(* Logix 5000 project; controller IPG_2332_07A 1769-L16ER-BB1B rev 34.12; software revision 34.01; part 3 of 4 *)
(* tags used below, declared in another part *)
   Axis_Controller : udt_Zaber_Axis;
   Flash_320mS : BOOL;
   Flash_640mS : BOOL;
   p_Alarmed_Time : String_15;
   p_All_Axis_Home : DINT;
   p_AOI_Cycle_Times : AOI_Cycle_Times;
   p_ASCII_RXID : DINT;
   p_ASCII_TXID : COUNTER;
   p_Axis_ONS : DINT;
   p_Barcode_results_Count_prev : DINT;
   p_BarcodeDone : BOOL;
   p_Cassette_Data : DINT;
   p_Cassette_Data_String : STRING;
   p_CassetteGripper_OUT : BOOL;
   p_CassetteRelease_IN : BOOL;   // Foot Switch
   p_Control : udt_Machine_Control_V2;   // Main Control
   p_Data_Reset : BOOL;
   p_DispenseStart_OUT : BOOL;
   p_DispenseTime : REAL;
   p_Downtime : String_15;
   p_FerruleGripper_OUT : BOOL;
   p_FiberAxis : udt_Zaber_Axis;
   p_FiberAxis_FinalMove_Done : BOOL;
   p_FiberAxis_FinalMoveRel : BOOL;
   p_FiberAxis_FindPos : udt_Station_Sequence;
   p_FiberAxis_InitialMove_Done : BOOL;
   p_FiberAxis_InitialMoveRel : BOOL;
   p_FiberAxis_Move_01_String : STRING;
   p_FiberAxis_Move_02_String : STRING;
   p_FiberGripper_OUT : BOOL;
   p_LED_Ramp : BOOL;
   p_LifeTime_Part_Counter : DINT;
   p_MirrorAxis : udt_Zaber_Axis;
   p_Part_Counter : DINT;
   p_PBLight_Amber_OUT : BOOL;
   p_PBLight_Green_OUT : BOOL;
   p_PBLight_Red_OUT : BOOL;
   p_Sequence : udt_Station_Sequence;
   p_StackLight_Amber_OUT : BOOL;
   p_StackLight_Green_OUT : BOOL;
   p_StackLight_Red_OUT : BOOL;
   p_SyringeAxis : udt_Zaber_Axis;
   p_Uptime : String_15;
   p_Waiting : BOOL;
   p_Waiting_Time : String_15;
   Debug_SDF : DINT;
(* MainProgram_10Ms, continued *)

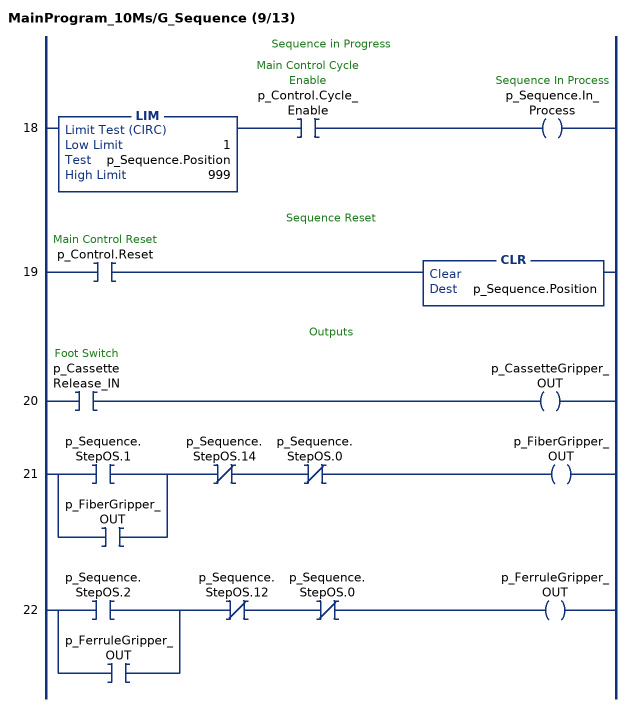
   [picture p43: MainProgram_10Ms/G_Sequence rungs 18-22]
   // Sequence in Progress
   18: LIM(1,p_Sequence.Position,999)XIC(p_Control.Cycle_Enable)OTE(p_Sequence.In_Process);
   // Sequence Reset
   19: XIC(p_Control.Reset)CLR(p_Sequence.Position);
   // Outputs
   20: XIC(p_CassetteRelease_IN)OTE(p_CassetteGripper_OUT);
   21: [XIC(p_Sequence.StepOS.1) ,XIC(p_FiberGripper_OUT) ]XIO(p_Sequence.StepOS.14)XIO(p_Sequence.StepOS.0)OTE(p_FiberGripper_OUT);
   22: [XIC(p_Sequence.StepOS.2) ,XIC(p_FerruleGripper_OUT) ]XIO(p_Sequence.StepOS.12)XIO(p_Sequence.StepOS.0)OTE(p_FerruleGripper_OUT);
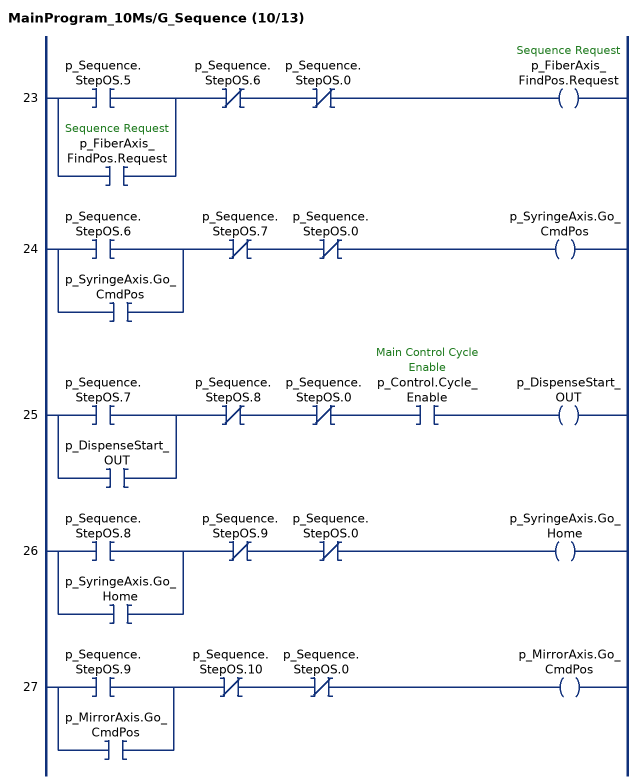
   23: [XIC(p_Sequence.StepOS.5) ,XIC(p_FiberAxis_FindPos.Request) ]XIO(p_Sequence.StepOS.6)XIO(p_Sequence.StepOS.0)OTE(p_FiberAxis_FindPos.Request);
   24: [XIC(p_Sequence.StepOS.6) ,XIC(p_SyringeAxis.Go_CmdPos) ]XIO(p_Sequence.StepOS.7)XIO(p_Sequence.StepOS.0)OTE(p_SyringeAxis.Go_CmdPos);
   25: [XIC(p_Sequence.StepOS.7) ,XIC(p_DispenseStart_OUT) ]XIO(p_Sequence.StepOS.8)XIO(p_Sequence.StepOS.0)XIC(p_Control.Cycle_Enable)OTE(p_DispenseStart_OUT);
   26: [XIC(p_Sequence.StepOS.8) ,XIC(p_SyringeAxis.Go_Home) ]XIO(p_Sequence.StepOS.9)XIO(p_Sequence.StepOS.0)OTE(p_SyringeAxis.Go_Home);
   27: [XIC(p_Sequence.StepOS.9) ,XIC(p_MirrorAxis.Go_CmdPos) ]XIO(p_Sequence.StepOS.10)XIO(p_Sequence.StepOS.0)OTE(p_MirrorAxis.Go_CmdPos);
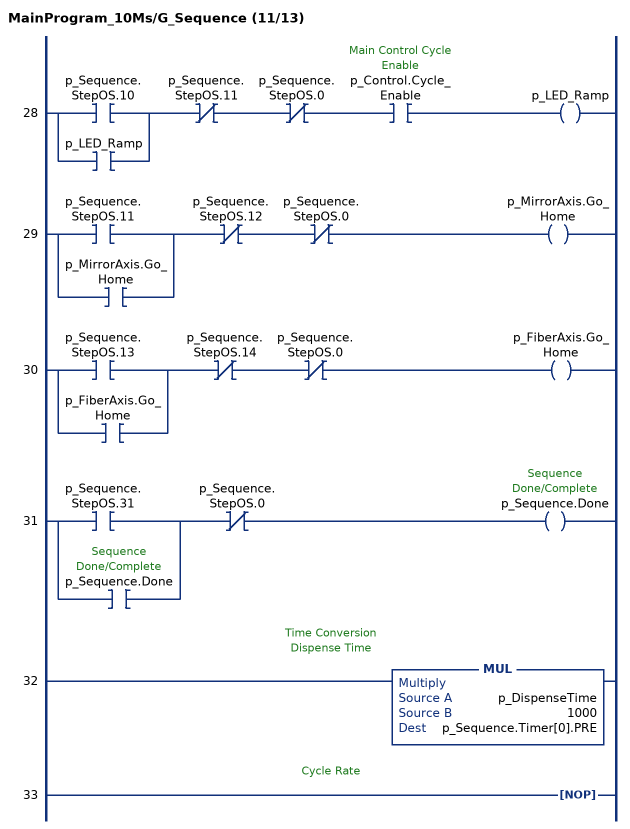
   28: [XIC(p_Sequence.StepOS.10) ,XIC(p_LED_Ramp) ]XIO(p_Sequence.StepOS.11)XIO(p_Sequence.StepOS.0)XIC(p_Control.Cycle_Enable)OTE(p_LED_Ramp);
   29: [XIC(p_Sequence.StepOS.11) ,XIC(p_MirrorAxis.Go_Home) ]XIO(p_Sequence.StepOS.12)XIO(p_Sequence.StepOS.0)OTE(p_MirrorAxis.Go_Home);
   30: [XIC(p_Sequence.StepOS.13) ,XIC(p_FiberAxis.Go_Home) ]XIO(p_Sequence.StepOS.14)XIO(p_Sequence.StepOS.0)OTE(p_FiberAxis.Go_Home);
   31: [XIC(p_Sequence.StepOS.31) ,XIC(p_Sequence.Done) ]XIO(p_Sequence.StepOS.0)OTE(p_Sequence.Done);
   // Time Conversion
   // Dispense Time
   32: MUL(p_DispenseTime,1000,p_Sequence.Timer[0].PRE);
   // Cycle Rate
   33: NOP();
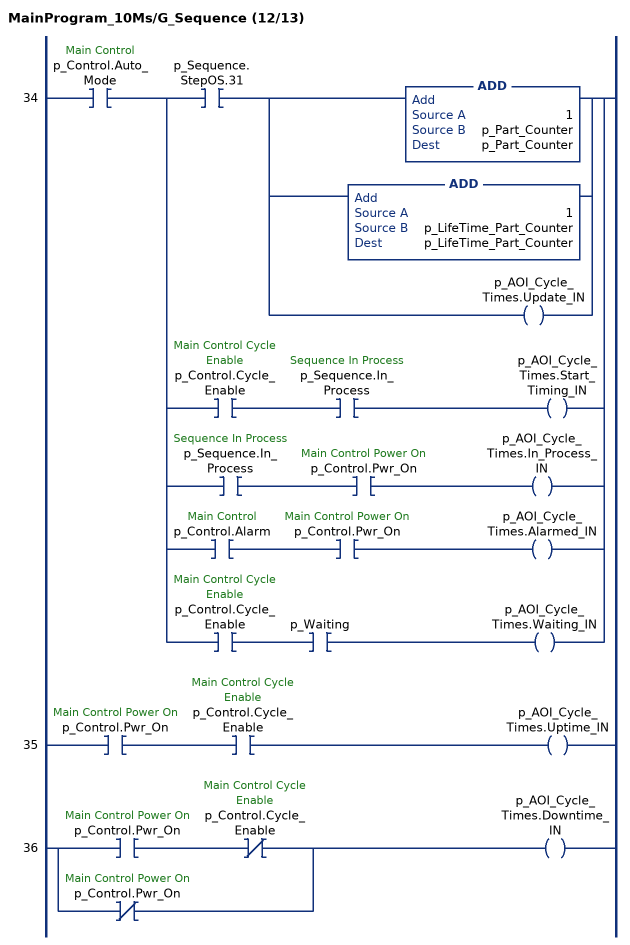
   34: XIC(p_Control.Auto_Mode)[XIC(p_Sequence.StepOS.31) [ADD(1,p_Part_Counter,p_Part_Counter) ,ADD(1,p_LifeTime_Part_Counter,p_LifeTime_Part_Counter) ,OTE(p_AOI_Cycle_Times.Update_IN) ] ,XIC(p_Control.Cycle_Enable) XIC(p_Sequence.In_Process) OTE(p_AOI_Cycle_Times.Start_Timing_IN) ,XIC(p_Sequence.In_Process) XIC(p_Control.Pwr_On) OTE(p_AOI_Cycle_Times.In_Process_IN) ,XIC(p_Control.Alarm) XIC(p_Control.Pwr_On) OTE(p_AOI_Cycle_Times.Alarmed_IN) ,XIC(p_Control.Cycle_Enable) XIC(p_Waiting) OTE(p_AOI_Cycle_Times.Waiting_IN) ];
   35: XIC(p_Control.Pwr_On)XIC(p_Control.Cycle_Enable)OTE(p_AOI_Cycle_Times.Uptime_IN);
   36: [XIC(p_Control.Pwr_On) XIO(p_Control.Cycle_Enable) ,XIO(p_Control.Pwr_On) ]OTE(p_AOI_Cycle_Times.Downtime_IN);
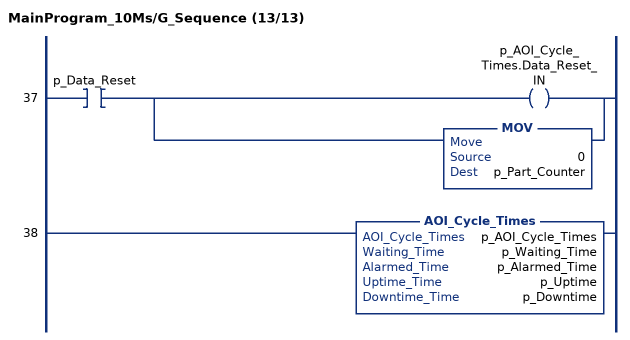
   37: XIC(p_Data_Reset)[OTE(p_AOI_Cycle_Times.Data_Reset_IN) ,MOV(0,p_Part_Counter) ];
   38: AOI_Cycle_Times(p_AOI_Cycle_Times,p_Waiting_Time,p_Alarmed_Time,p_Uptime,p_Downtime);
END_ROUTINE

ROUTINE H_QR_Reader   (* ladder *)
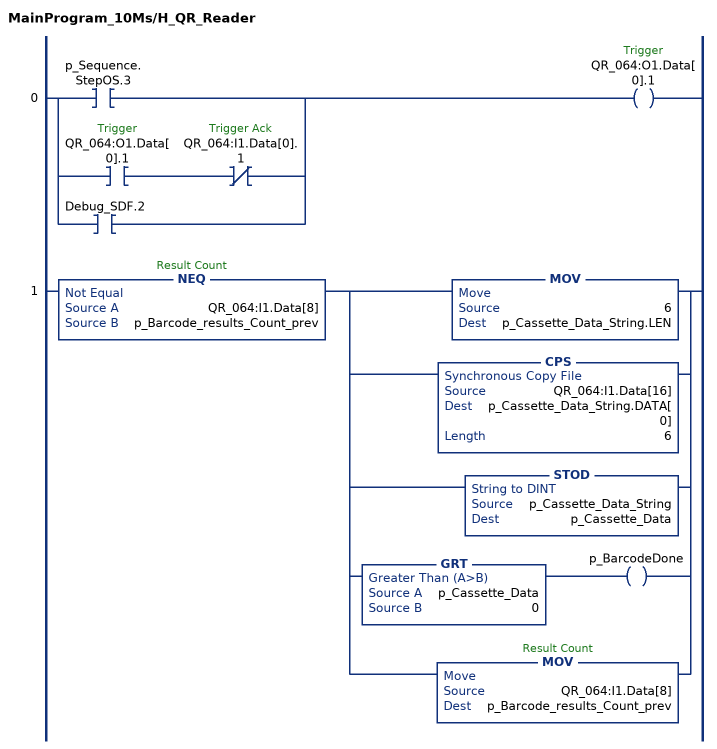
   0: [XIC(p_Sequence.StepOS.3) ,XIC(QR_064:O1.Data[0].1) XIO(QR_064:I1.Data[0].1) ,XIC(Debug_SDF.2) ]OTE(QR_064:O1.Data[0].1);
   1: NEQ(QR_064:I1.Data[8],p_Barcode_results_Count_prev)[MOV(6,p_Cassette_Data_String.LEN) ,CPS(QR_064:I1.Data[16],p_Cassette_Data_String.DATA[0],6) ,STOD(p_Cassette_Data_String,p_Cassette_Data) ,GRT(p_Cassette_Data,0) OTE(p_BarcodeDone) ,MOV(QR_064:I1.Data[8],p_Barcode_results_Count_prev) ];
END_ROUTINE

ROUTINE I_Database_Com   (* ladder *)
   0: NOP();
END_ROUTINE

ROUTINE J_LightStack_PBLight   (* ladder *)
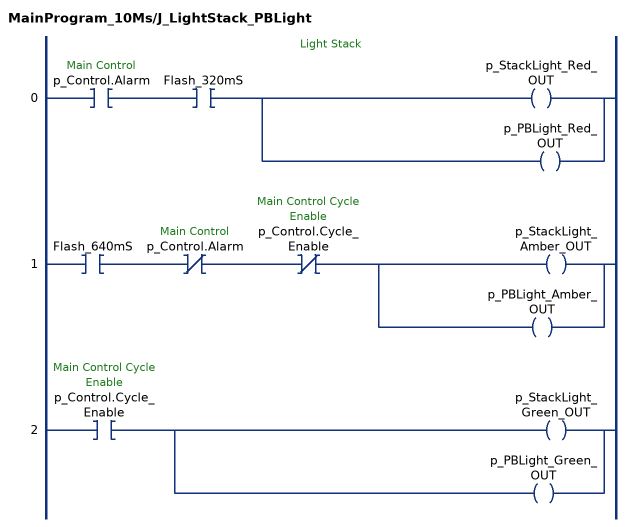
   // Light Stack
   0: XIC(p_Control.Alarm)XIC(Flash_320mS)[OTE(p_StackLight_Red_OUT) ,OTE(p_PBLight_Red_OUT) ];
   1: XIC(Flash_640mS)XIO(p_Control.Alarm)XIO(p_Control.Cycle_Enable)[OTE(p_StackLight_Amber_OUT) ,OTE(p_PBLight_Amber_OUT) ];
   2: XIC(p_Control.Cycle_Enable)[OTE(p_StackLight_Green_OUT) ,OTE(p_PBLight_Green_OUT) ];
END_ROUTINE

ROUTINE K_AxisControl   (* ladder *)
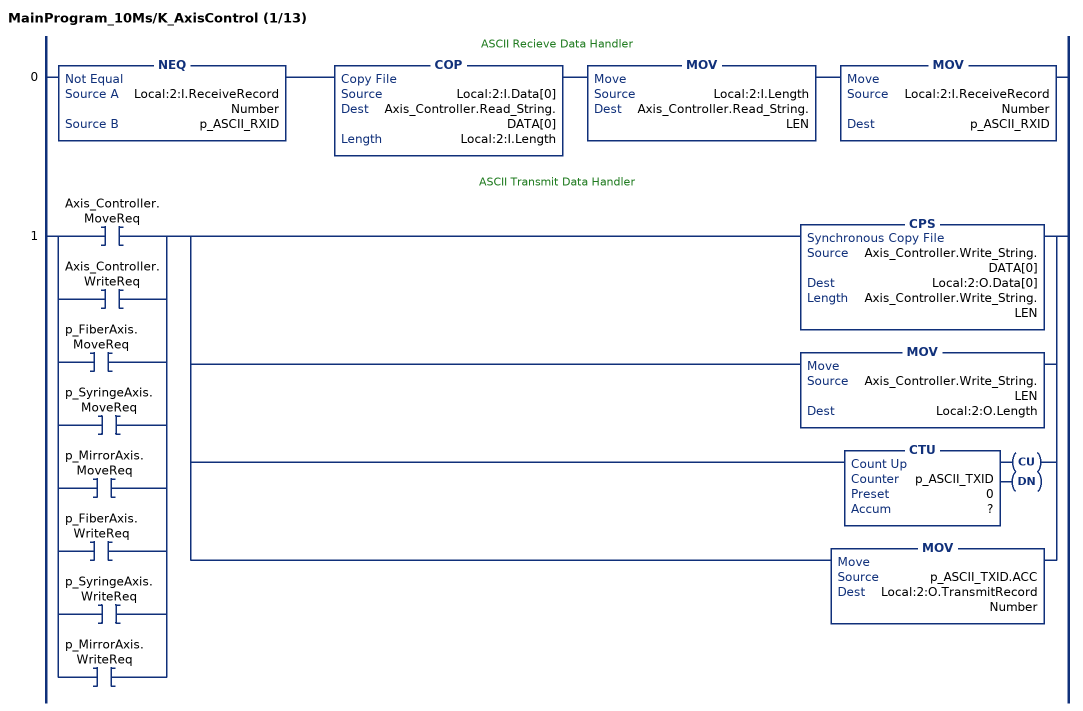
   // ASCII Recieve Data Handler
   0: NEQ(Local:2:I.ReceiveRecordNumber,p_ASCII_RXID)COP(Local:2:I.Data[0],Axis_Controller.Read_String.DATA[0],Local:2:I.Length)MOV(Local:2:I.Length,Axis_Controller.Read_String.LEN)MOV(Local:2:I.ReceiveRecordNumber,p_ASCII_RXID);
   // ASCII Transmit Data Handler
   1: [XIC(Axis_Controller.MoveReq) ,XIC(Axis_Controller.WriteReq) ,XIC(p_FiberAxis.MoveReq) ,XIC(p_SyringeAxis.MoveReq) ,XIC(p_MirrorAxis.MoveReq) ,XIC(p_FiberAxis.WriteReq) ,XIC(p_SyringeAxis.WriteReq) ,XIC(p_MirrorAxis.WriteReq) ][CPS(Axis_Controller.Write_String.DATA[0],Local:2:O.Data[0],Axis_Controller.Write_String.LEN) ,MOV(Axis_Controller.Write_String.LEN,Local:2:O.Length) ,CTU(p_ASCII_TXID,?,?) ,MOV(p_ASCII_TXID.ACC,Local:2:O.TransmitRecordNumber) ];
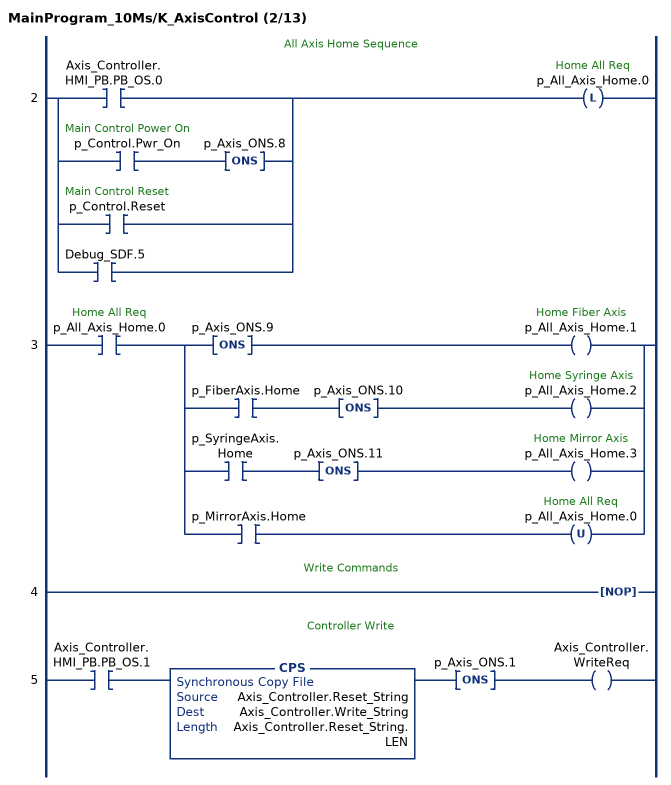
   // All Axis Home Sequence
   2: [XIC(Axis_Controller.HMI_PB.PB_OS.0) ,XIC(p_Control.Pwr_On) ONS(p_Axis_ONS.8) ,XIC(p_Control.Reset) ,XIC(Debug_SDF.5) ]OTL(p_All_Axis_Home.0);
   3: XIC(p_All_Axis_Home.0)[ONS(p_Axis_ONS.9) OTE(p_All_Axis_Home.1) ,XIC(p_FiberAxis.Home) ONS(p_Axis_ONS.10) OTE(p_All_Axis_Home.2) ,XIC(p_SyringeAxis.Home) ONS(p_Axis_ONS.11) OTE(p_All_Axis_Home.3) ,XIC(p_MirrorAxis.Home) OTU(p_All_Axis_Home.0) ];
   // Write Commands
   4: NOP();
   // Controller Write
   5: XIC(Axis_Controller.HMI_PB.PB_OS.1)CPS(Axis_Controller.Reset_String,Axis_Controller.Write_String,Axis_Controller.Reset_String.LEN)ONS(p_Axis_ONS.1)OTE(Axis_Controller.WriteReq);
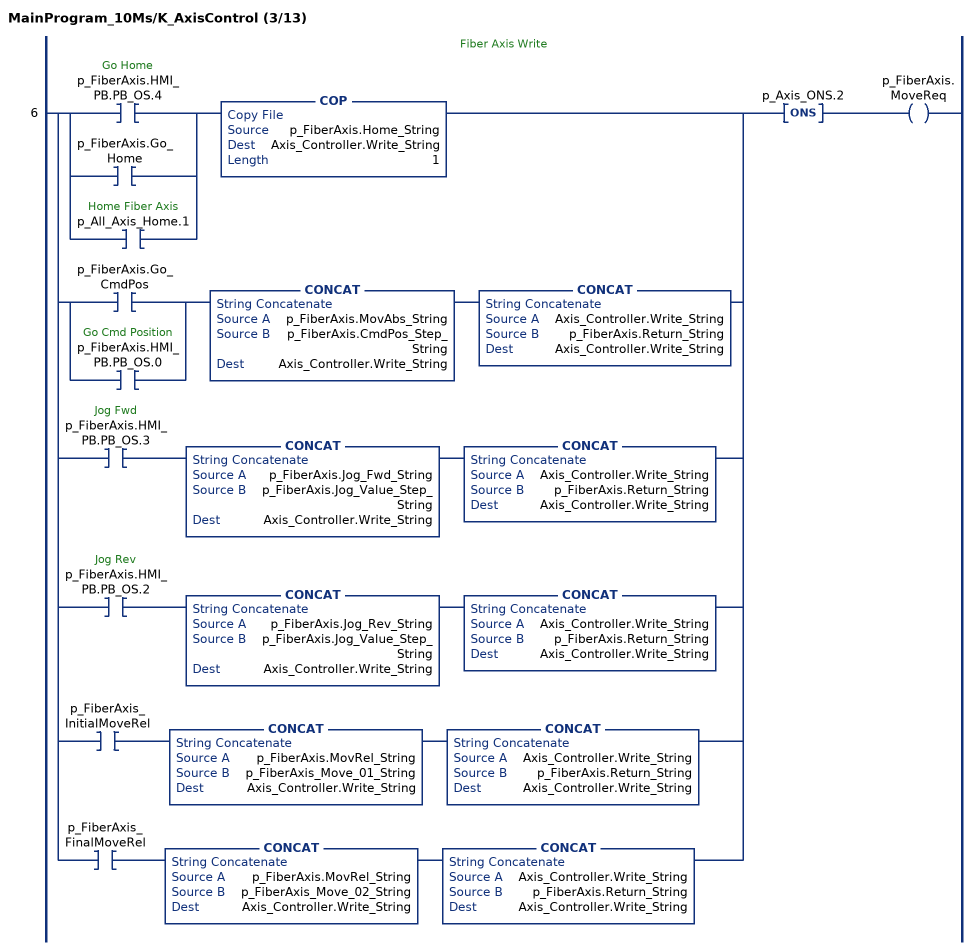
   // Fiber Axis Write
   6: [[XIC(p_FiberAxis.HMI_PB.PB_OS.4) ,XIC(p_FiberAxis.Go_Home) ,XIC(p_All_Axis_Home.1) ] COP(p_FiberAxis.Home_String,Axis_Controller.Write_String,1) ,[XIC(p_FiberAxis.Go_CmdPos) ,XIC(p_FiberAxis.HMI_PB.PB_OS.0) ] CONCAT(p_FiberAxis.MovAbs_String,p_FiberAxis.CmdPos_Step_String,Axis_Controller.Write_String) CONCAT(Axis_Controller.Write_String,p_FiberAxis.Return_String,Axis_Controller.Write_String) ,XIC(p_FiberAxis.HMI_PB.PB_OS.3) CONCAT(p_FiberAxis.Jog_Fwd_String,p_FiberAxis.Jog_Value_Step_String,Axis_Controller.Write_String) CONCAT(Axis_Controller.Write_String,p_FiberAxis.Return_String,Axis_Controller.Write_String) ,XIC(p_FiberAxis.HMI_PB.PB_OS.2) CONCAT(p_FiberAxis.Jog_Rev_String,p_FiberAxis.Jog_Value_Step_String,Axis_Controller.Write_String) CONCAT(Axis_Controller.Write_String,p_FiberAxis.Return_String,Axis_Controller.Write_String) ,XIC(p_FiberAxis_InitialMoveRel) CONCAT(p_FiberAxis.MovRel_String,p_FiberAxis_Move_01_String,Axis_Controller.Write_String) CONCAT(Axis_Controller.Write_String,p_FiberAxis.Return_String,Axis_Controller.Write_String) ,XIC(p_FiberAxis_FinalMoveRel) CONCAT(p_FiberAxis.MovRel_String,p_FiberAxis_Move_02_String,Axis_Controller.Write_String) CONCAT(Axis_Controller.Write_String,p_FiberAxis.Return_String,Axis_Controller.Write_String) ]ONS(p_Axis_ONS.2)OTE(p_FiberAxis.MoveReq);
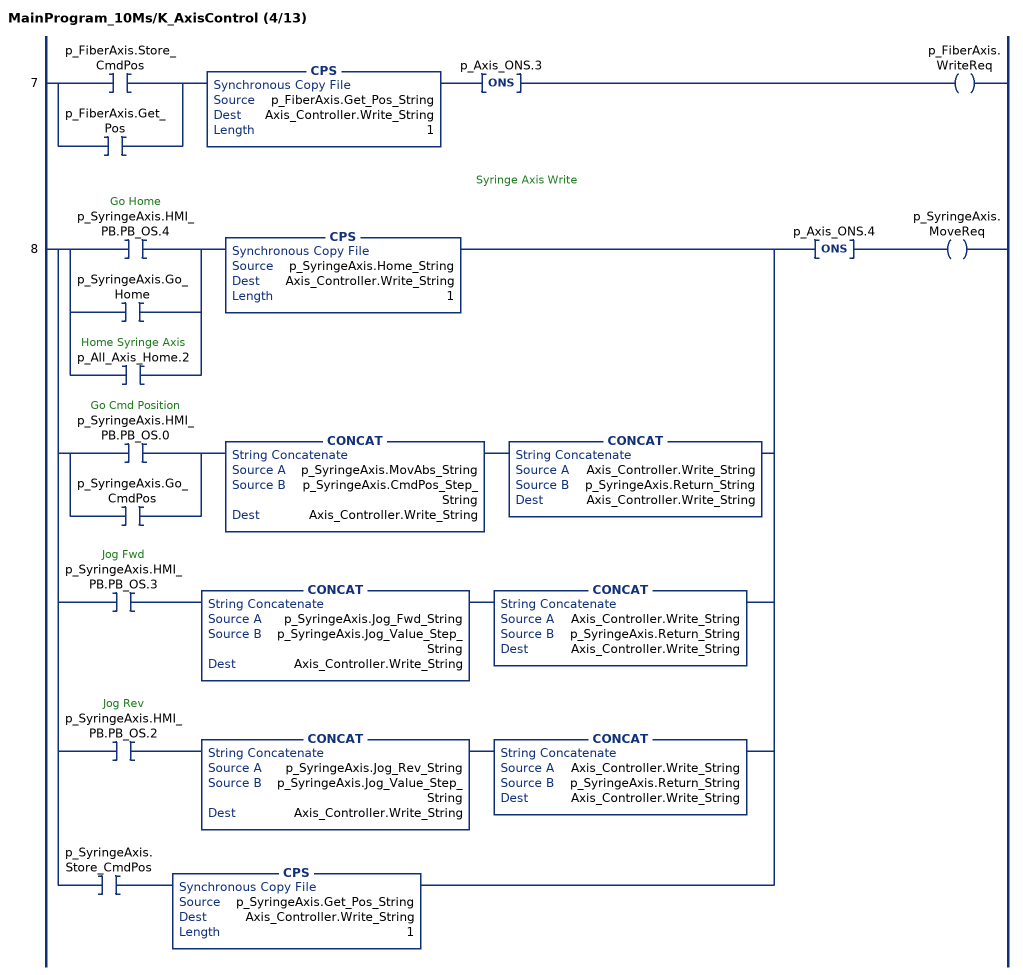
   7: [XIC(p_FiberAxis.Store_CmdPos) ,XIC(p_FiberAxis.Get_Pos) ]CPS(p_FiberAxis.Get_Pos_String,Axis_Controller.Write_String,1)ONS(p_Axis_ONS.3)OTE(p_FiberAxis.WriteReq);
   // Syringe Axis Write
   8: [[XIC(p_SyringeAxis.HMI_PB.PB_OS.4) ,XIC(p_SyringeAxis.Go_Home) ,XIC(p_All_Axis_Home.2) ] CPS(p_SyringeAxis.Home_String,Axis_Controller.Write_String,1) ,[XIC(p_SyringeAxis.HMI_PB.PB_OS.0) ,XIC(p_SyringeAxis.Go_CmdPos) ] CONCAT(p_SyringeAxis.MovAbs_String,p_SyringeAxis.CmdPos_Step_String,Axis_Controller.Write_String) CONCAT(Axis_Controller.Write_String,p_SyringeAxis.Return_String,Axis_Controller.Write_String) ,XIC(p_SyringeAxis.HMI_PB.PB_OS.3) CONCAT(p_SyringeAxis.Jog_Fwd_String,p_SyringeAxis.Jog_Value_Step_String,Axis_Controller.Write_String) CONCAT(Axis_Controller.Write_String,p_SyringeAxis.Return_String,Axis_Controller.Write_String) ,XIC(p_SyringeAxis.HMI_PB.PB_OS.2) CONCAT(p_SyringeAxis.Jog_Rev_String,p_SyringeAxis.Jog_Value_Step_String,Axis_Controller.Write_String) CONCAT(Axis_Controller.Write_String,p_SyringeAxis.Return_String,Axis_Controller.Write_String) ,XIC(p_SyringeAxis.Store_CmdPos) CPS(p_SyringeAxis.Get_Pos_String,Axis_Controller.Write_String,1) ]ONS(p_Axis_ONS.4)OTE(p_SyringeAxis.MoveReq);
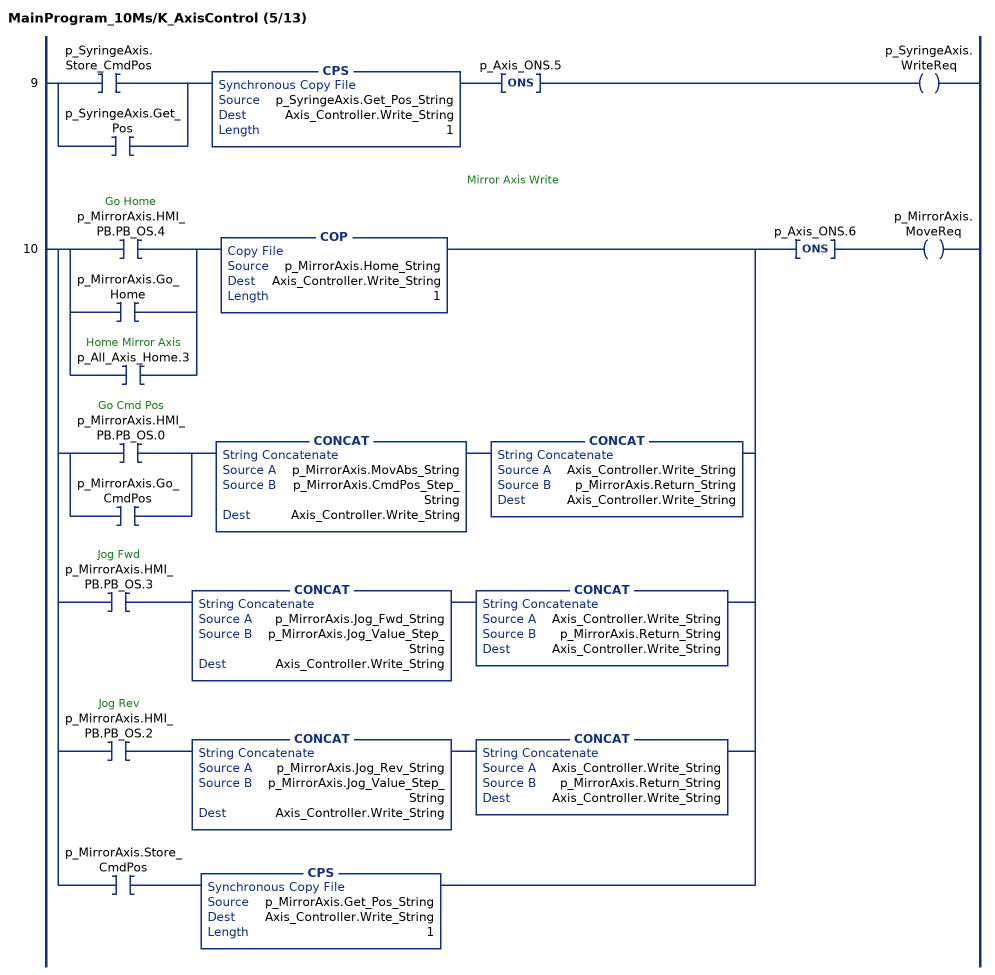
   9: [XIC(p_SyringeAxis.Store_CmdPos) ,XIC(p_SyringeAxis.Get_Pos) ]CPS(p_SyringeAxis.Get_Pos_String,Axis_Controller.Write_String,1)ONS(p_Axis_ONS.5)OTE(p_SyringeAxis.WriteReq);
   // Mirror Axis Write
   10: [[XIC(p_MirrorAxis.HMI_PB.PB_OS.4) ,XIC(p_MirrorAxis.Go_Home) ,XIC(p_All_Axis_Home.3) ] COP(p_MirrorAxis.Home_String,Axis_Controller.Write_String,1) ,[XIC(p_MirrorAxis.HMI_PB.PB_OS.0) ,XIC(p_MirrorAxis.Go_CmdPos) ] CONCAT(p_MirrorAxis.MovAbs_String,p_MirrorAxis.CmdPos_Step_String,Axis_Controller.Write_String) CONCAT(Axis_Controller.Write_String,p_MirrorAxis.Return_String,Axis_Controller.Write_String) ,XIC(p_MirrorAxis.HMI_PB.PB_OS.3) CONCAT(p_MirrorAxis.Jog_Fwd_String,p_MirrorAxis.Jog_Value_Step_String,Axis_Controller.Write_String) CONCAT(Axis_Controller.Write_String,p_MirrorAxis.Return_String,Axis_Controller.Write_String) ,XIC(p_MirrorAxis.HMI_PB.PB_OS.2) CONCAT(p_MirrorAxis.Jog_Rev_String,p_MirrorAxis.Jog_Value_Step_String,Axis_Controller.Write_String) CONCAT(Axis_Controller.Write_String,p_MirrorAxis.Return_String,Axis_Controller.Write_String) ,XIC(p_MirrorAxis.Store_CmdPos) CPS(p_MirrorAxis.Get_Pos_String,Axis_Controller.Write_String,1) ]ONS(p_Axis_ONS.6)OTE(p_MirrorAxis.MoveReq);
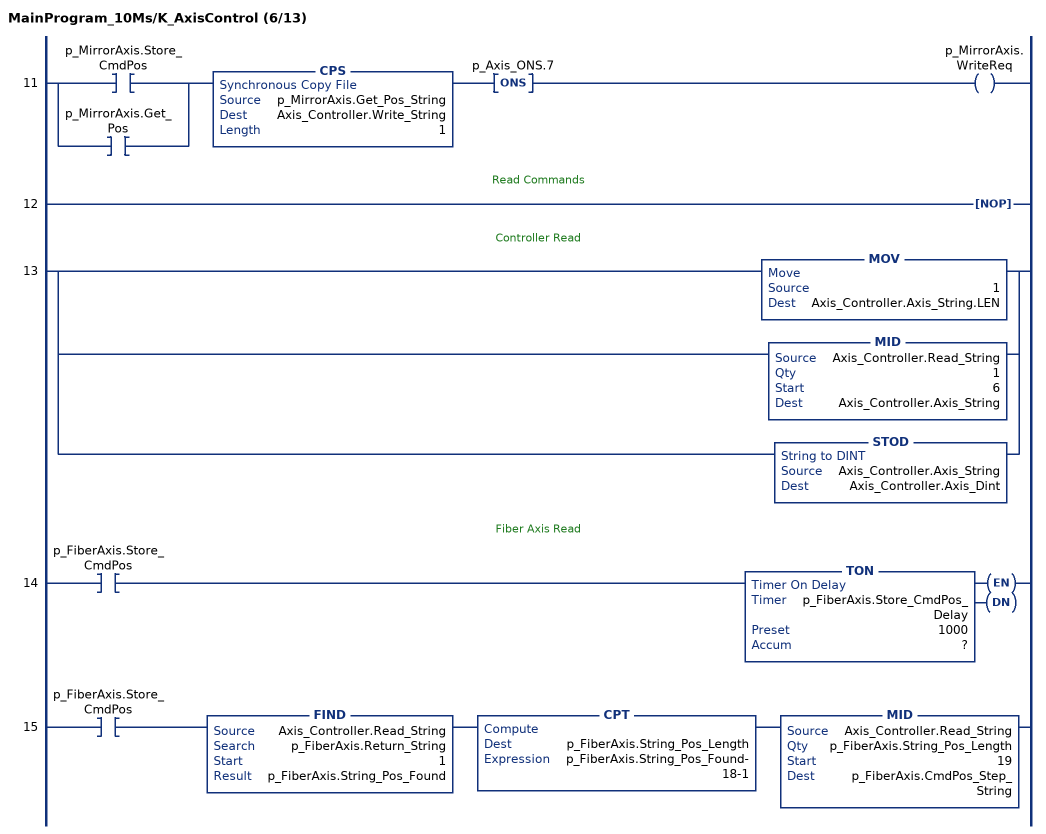
   11: [XIC(p_MirrorAxis.Store_CmdPos) ,XIC(p_MirrorAxis.Get_Pos) ]CPS(p_MirrorAxis.Get_Pos_String,Axis_Controller.Write_String,1)ONS(p_Axis_ONS.7)OTE(p_MirrorAxis.WriteReq);
   // Read Commands
   12: NOP();
   // Controller Read
   13: [MOV(1,Axis_Controller.Axis_String.LEN) ,MID(Axis_Controller.Read_String,1,6,Axis_Controller.Axis_String) ,STOD(Axis_Controller.Axis_String,Axis_Controller.Axis_Dint) ];
   // Fiber Axis Read
   14: XIC(p_FiberAxis.Store_CmdPos)TON(p_FiberAxis.Store_CmdPos_Delay,?,?);
   15: XIC(p_FiberAxis.Store_CmdPos)FIND(Axis_Controller.Read_String,p_FiberAxis.Return_String,1,p_FiberAxis.String_Pos_Found)CPT(p_FiberAxis.String_Pos_Length,p_FiberAxis.String_Pos_Found-18-1)MID(Axis_Controller.Read_String,p_FiberAxis.String_Pos_Length,19,p_FiberAxis.CmdPos_Step_String);
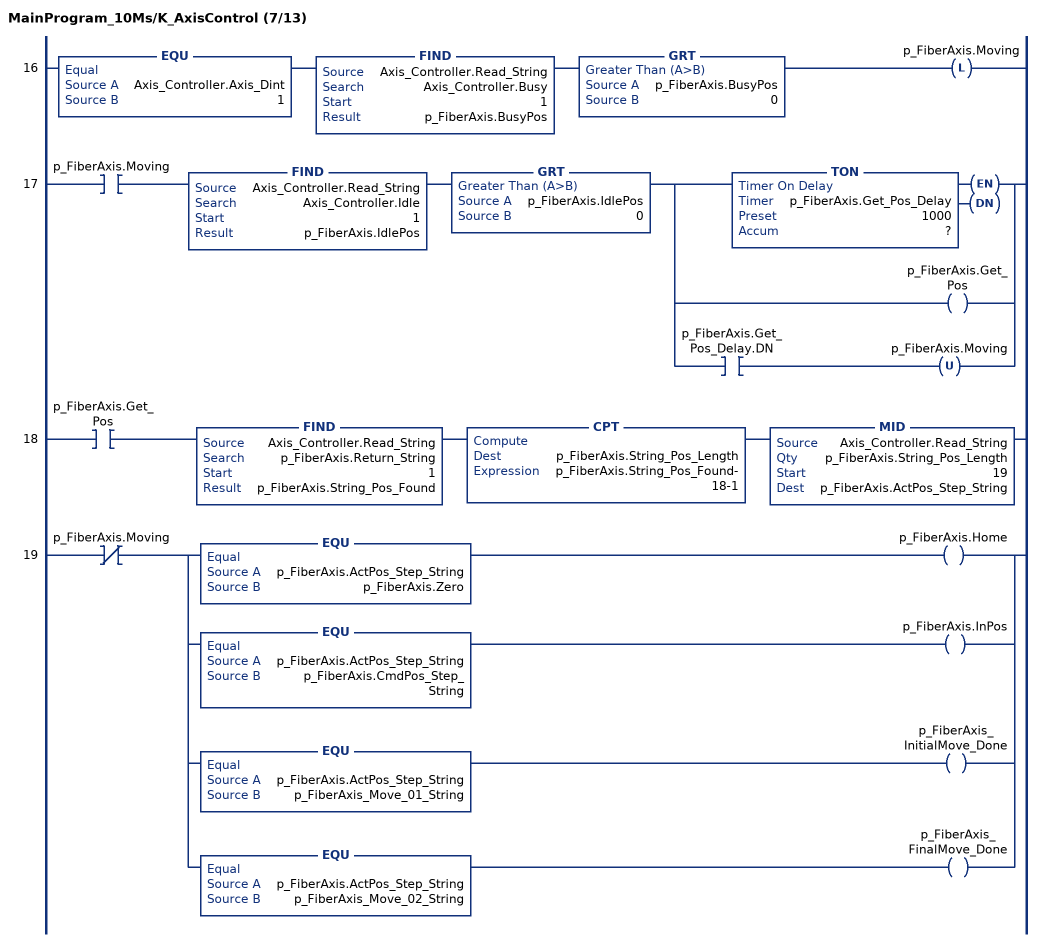
   16: EQU(Axis_Controller.Axis_Dint,1)FIND(Axis_Controller.Read_String,Axis_Controller.Busy,1,p_FiberAxis.BusyPos)GRT(p_FiberAxis.BusyPos,0)OTL(p_FiberAxis.Moving);
   17: XIC(p_FiberAxis.Moving)FIND(Axis_Controller.Read_String,Axis_Controller.Idle,1,p_FiberAxis.IdlePos)GRT(p_FiberAxis.IdlePos,0)[TON(p_FiberAxis.Get_Pos_Delay,?,?) ,OTE(p_FiberAxis.Get_Pos) ,XIC(p_FiberAxis.Get_Pos_Delay.DN) OTU(p_FiberAxis.Moving) ];
   18: XIC(p_FiberAxis.Get_Pos)FIND(Axis_Controller.Read_String,p_FiberAxis.Return_String,1,p_FiberAxis.String_Pos_Found)CPT(p_FiberAxis.String_Pos_Length,p_FiberAxis.String_Pos_Found-18-1)MID(Axis_Controller.Read_String,p_FiberAxis.String_Pos_Length,19,p_FiberAxis.ActPos_Step_String);
   19: XIO(p_FiberAxis.Moving)[EQU(p_FiberAxis.ActPos_Step_String,p_FiberAxis.Zero) OTE(p_FiberAxis.Home) ,EQU(p_FiberAxis.ActPos_Step_String,p_FiberAxis.CmdPos_Step_String) OTE(p_FiberAxis.InPos) ,EQU(p_FiberAxis.ActPos_Step_String,p_FiberAxis_Move_01_String) OTE(p_FiberAxis_InitialMove_Done) ,EQU(p_FiberAxis.ActPos_Step_String,p_FiberAxis_Move_02_String) OTE(p_FiberAxis_FinalMove_Done) ];
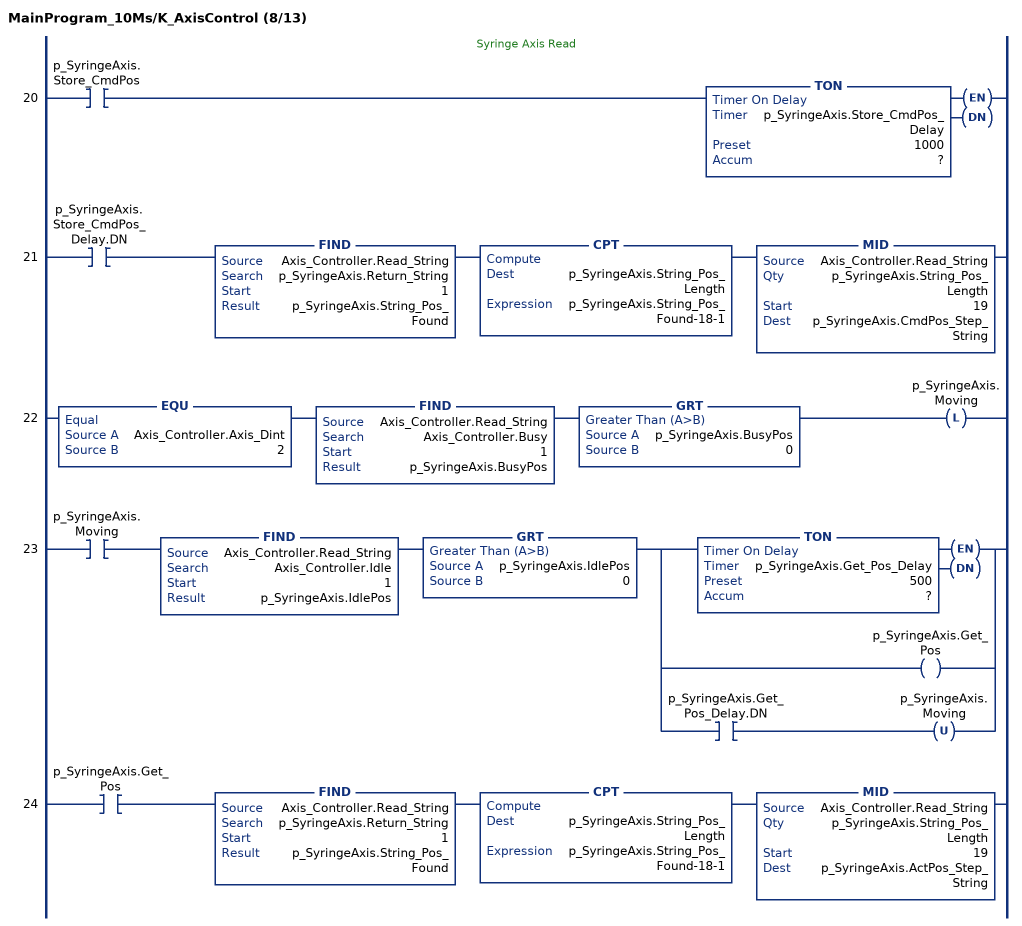
   // Syringe Axis Read
   20: XIC(p_SyringeAxis.Store_CmdPos)TON(p_SyringeAxis.Store_CmdPos_Delay,?,?);
   21: XIC(p_SyringeAxis.Store_CmdPos_Delay.DN)FIND(Axis_Controller.Read_String,p_SyringeAxis.Return_String,1,p_SyringeAxis.String_Pos_Found)CPT(p_SyringeAxis.String_Pos_Length,p_SyringeAxis.String_Pos_Found-18-1)MID(Axis_Controller.Read_String,p_SyringeAxis.String_Pos_Length,19,p_SyringeAxis.CmdPos_Step_String);
   22: EQU(Axis_Controller.Axis_Dint,2)FIND(Axis_Controller.Read_String,Axis_Controller.Busy,1,p_SyringeAxis.BusyPos)GRT(p_SyringeAxis.BusyPos,0)OTL(p_SyringeAxis.Moving);
   23: XIC(p_SyringeAxis.Moving)FIND(Axis_Controller.Read_String,Axis_Controller.Idle,1,p_SyringeAxis.IdlePos)GRT(p_SyringeAxis.IdlePos,0)[TON(p_SyringeAxis.Get_Pos_Delay,?,?) ,OTE(p_SyringeAxis.Get_Pos) ,XIC(p_SyringeAxis.Get_Pos_Delay.DN) OTU(p_SyringeAxis.Moving) ];
   24: XIC(p_SyringeAxis.Get_Pos)FIND(Axis_Controller.Read_String,p_SyringeAxis.Return_String,1,p_SyringeAxis.String_Pos_Found)CPT(p_SyringeAxis.String_Pos_Length,p_SyringeAxis.String_Pos_Found-18-1)MID(Axis_Controller.Read_String,p_SyringeAxis.String_Pos_Length,19,p_SyringeAxis.ActPos_Step_String);
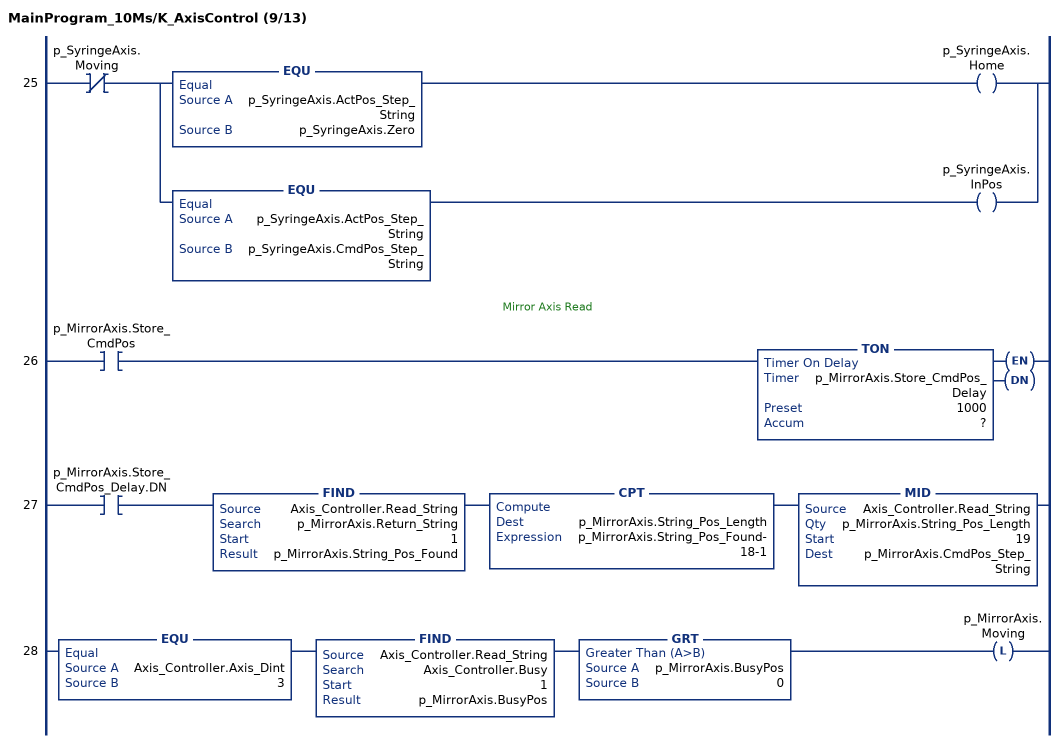
   25: XIO(p_SyringeAxis.Moving)[EQU(p_SyringeAxis.ActPos_Step_String,p_SyringeAxis.Zero) OTE(p_SyringeAxis.Home) ,EQU(p_SyringeAxis.ActPos_Step_String,p_SyringeAxis.CmdPos_Step_String) OTE(p_SyringeAxis.InPos) ];
   // Mirror Axis Read
   26: XIC(p_MirrorAxis.Store_CmdPos)TON(p_MirrorAxis.Store_CmdPos_Delay,?,?);
   27: XIC(p_MirrorAxis.Store_CmdPos_Delay.DN)FIND(Axis_Controller.Read_String,p_MirrorAxis.Return_String,1,p_MirrorAxis.String_Pos_Found)CPT(p_MirrorAxis.String_Pos_Length,p_MirrorAxis.String_Pos_Found-18-1)MID(Axis_Controller.Read_String,p_MirrorAxis.String_Pos_Length,19,p_MirrorAxis.CmdPos_Step_String);
   28: EQU(Axis_Controller.Axis_Dint,3)FIND(Axis_Controller.Read_String,Axis_Controller.Busy,1,p_MirrorAxis.BusyPos)GRT(p_MirrorAxis.BusyPos,0)OTL(p_MirrorAxis.Moving);
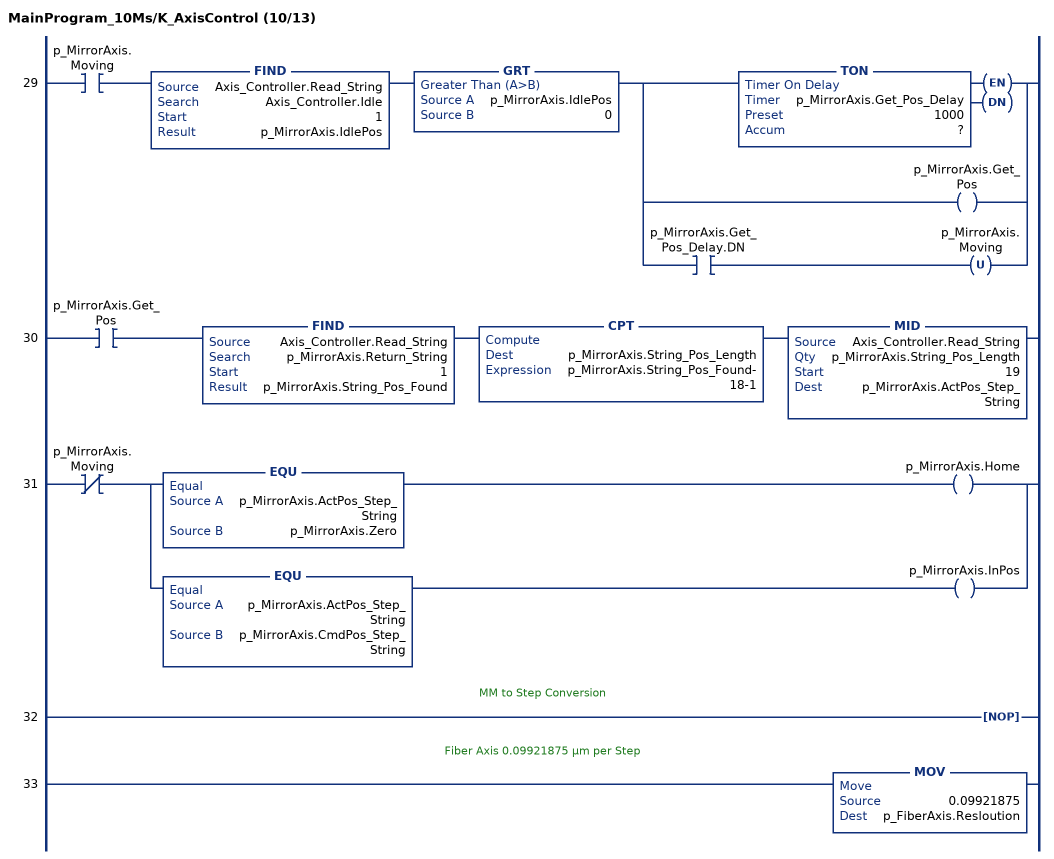
   29: XIC(p_MirrorAxis.Moving)FIND(Axis_Controller.Read_String,Axis_Controller.Idle,1,p_MirrorAxis.IdlePos)GRT(p_MirrorAxis.IdlePos,0)[TON(p_MirrorAxis.Get_Pos_Delay,?,?) ,OTE(p_MirrorAxis.Get_Pos) ,XIC(p_MirrorAxis.Get_Pos_Delay.DN) OTU(p_MirrorAxis.Moving) ];
   30: XIC(p_MirrorAxis.Get_Pos)FIND(Axis_Controller.Read_String,p_MirrorAxis.Return_String,1,p_MirrorAxis.String_Pos_Found)CPT(p_MirrorAxis.String_Pos_Length,p_MirrorAxis.String_Pos_Found-18-1)MID(Axis_Controller.Read_String,p_MirrorAxis.String_Pos_Length,19,p_MirrorAxis.ActPos_Step_String);
   31: XIO(p_MirrorAxis.Moving)[EQU(p_MirrorAxis.ActPos_Step_String,p_MirrorAxis.Zero) OTE(p_MirrorAxis.Home) ,EQU(p_MirrorAxis.ActPos_Step_String,p_MirrorAxis.CmdPos_Step_String) OTE(p_MirrorAxis.InPos) ];
   // MM to Step Conversion
   32: NOP();
   // Fiber Axis 0.09921875 µm per Step
   33: MOV(0.09921875,p_FiberAxis.Resloution);
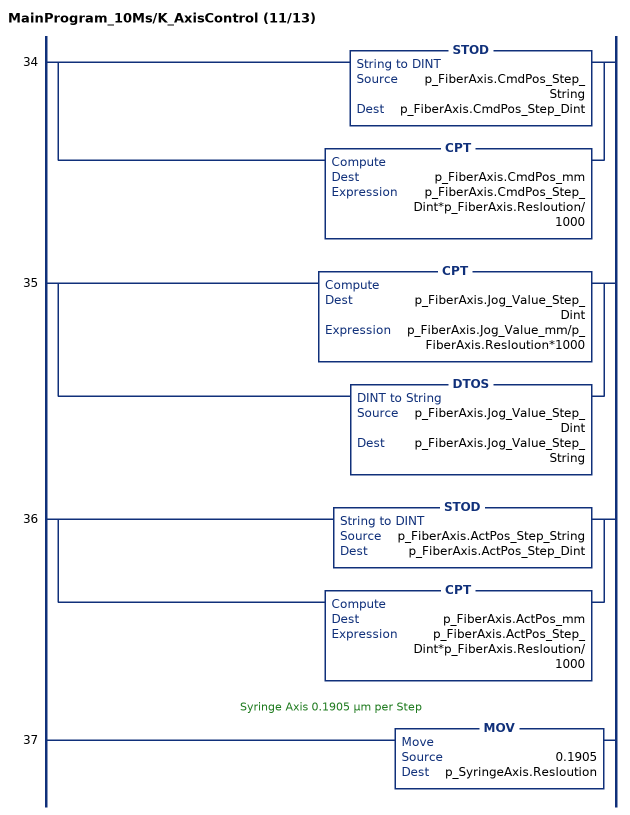
   34: [STOD(p_FiberAxis.CmdPos_Step_String,p_FiberAxis.CmdPos_Step_Dint) ,CPT(p_FiberAxis.CmdPos_mm,p_FiberAxis.CmdPos_Step_Dint*p_FiberAxis.Resloution/1000) ];
   35: [CPT(p_FiberAxis.Jog_Value_Step_Dint,p_FiberAxis.Jog_Value_mm/p_FiberAxis.Resloution*1000) ,DTOS(p_FiberAxis.Jog_Value_Step_Dint,p_FiberAxis.Jog_Value_Step_String) ];
   36: [STOD(p_FiberAxis.ActPos_Step_String,p_FiberAxis.ActPos_Step_Dint) ,CPT(p_FiberAxis.ActPos_mm,p_FiberAxis.ActPos_Step_Dint*p_FiberAxis.Resloution/1000) ];
   // Syringe Axis 0.1905 µm per Step
   37: MOV(0.1905,p_SyringeAxis.Resloution);
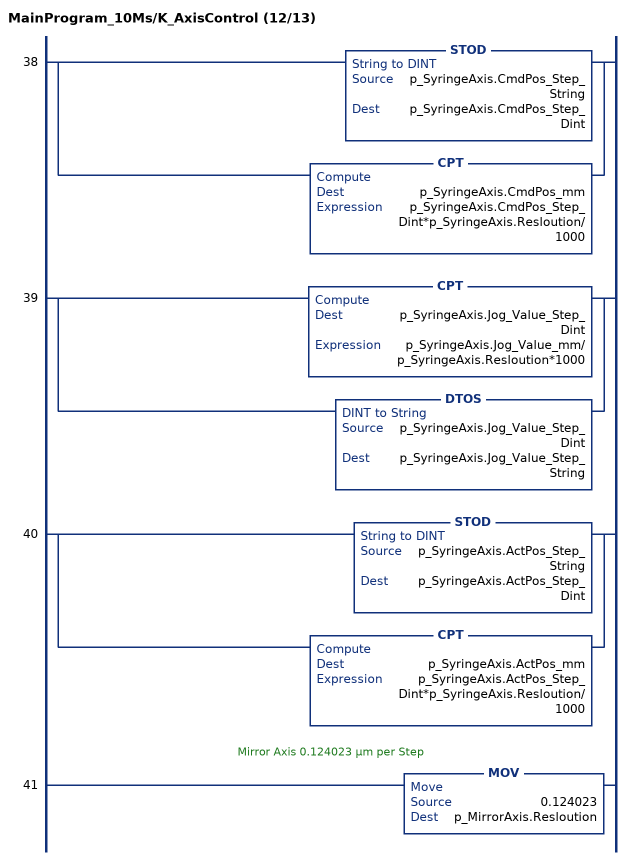
   38: [STOD(p_SyringeAxis.CmdPos_Step_String,p_SyringeAxis.CmdPos_Step_Dint) ,CPT(p_SyringeAxis.CmdPos_mm,p_SyringeAxis.CmdPos_Step_Dint*p_SyringeAxis.Resloution/1000) ];
   39: [CPT(p_SyringeAxis.Jog_Value_Step_Dint,p_SyringeAxis.Jog_Value_mm/p_SyringeAxis.Resloution*1000) ,DTOS(p_SyringeAxis.Jog_Value_Step_Dint,p_SyringeAxis.Jog_Value_Step_String) ];
   40: [STOD(p_SyringeAxis.ActPos_Step_String,p_SyringeAxis.ActPos_Step_Dint) ,CPT(p_SyringeAxis.ActPos_mm,p_SyringeAxis.ActPos_Step_Dint*p_SyringeAxis.Resloution/1000) ];
   // Mirror Axis 0.124023 µm per Step
   41: MOV(0.124023,p_MirrorAxis.Resloution);
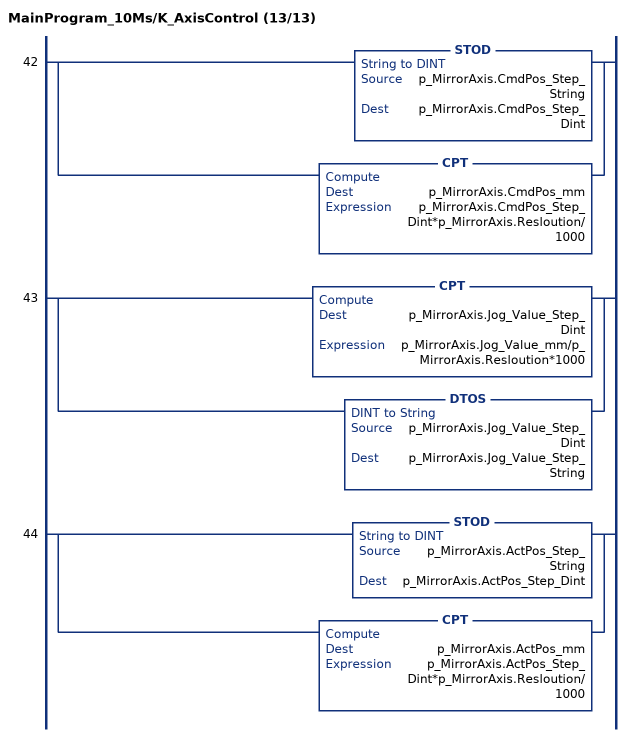
   42: [STOD(p_MirrorAxis.CmdPos_Step_String,p_MirrorAxis.CmdPos_Step_Dint) ,CPT(p_MirrorAxis.CmdPos_mm,p_MirrorAxis.CmdPos_Step_Dint*p_MirrorAxis.Resloution/1000) ];
   43: [CPT(p_MirrorAxis.Jog_Value_Step_Dint,p_MirrorAxis.Jog_Value_mm/p_MirrorAxis.Resloution*1000) ,DTOS(p_MirrorAxis.Jog_Value_Step_Dint,p_MirrorAxis.Jog_Value_Step_String) ];
   44: [STOD(p_MirrorAxis.ActPos_Step_String,p_MirrorAxis.ActPos_Step_Dint) ,CPT(p_MirrorAxis.ActPos_mm,p_MirrorAxis.ActPos_Step_Dint*p_MirrorAxis.Resloution/1000) ];
END_ROUTINE
